(* CODESYS project filling_station.ecp

Project tree, tasks and I/O mapping:
  GenericDummyMasterDevice : Generic Master, WAGO, order no. None, version 1.0.0.0
  PFC200_CS_2ETH_RS : 750-8202 PFC200 2ETH RS, WAGO, order no. 0750-8202, version 1.4.1.22
    application Application
      libraries: 
      task PLC_Task (cyclic, interval t#10ms, priority 14) calls PLC_PRG
      program PLC_PRG [ST]
    DeviceAdapter
    Kbus : Kbus, WAGO, version 1.3.0.0
        unmapped channels: K-BUS diagnostics
      _8_DO_Generic : 075x-8DO, WAGO, order no. 075x-8DO, version 0.0.0.11
          settings: K-BUS Module slot index = 1
          unmapped channels: _OUT
        DeviceAdapter
      _4_AI_0_10V_DC_s_e : 0750-0459, WAGO, order no. 0750-0459, version 0.0.0.11
          settings: K-BUS Module slot index = 2
          unmapped channels: _IW 1, _IW 2, _IW 3, _IW 4
        DeviceAdapter
      _2_AI_4_20mA_Diff_Measurement_Input : 0750-0492, WAGO, order no. 0750-0492, version 0.0.0.7
          settings: K-BUS Module slot index = 3
          unmapped channels: _IW 1, _IW 2
        DeviceAdapter
    MODBUS
      MODBUS : MODBUS, WAGO, order no. n/a, version 1.1.1.13
    Serial
      COM1 : COM1, WAGO, version 0.0.0.19
*)

// PFC200_CS_2ETH_RS/Application/PLC_PRG
PROGRAM PLC_PRG
VAR
END_VAR

END_PROGRAM
